                          .stSerial1.stComOut.D[0]  		:= TIIB[PCM A (EP6002-0002)]^COM RxPDO-Map Outputs Channel 1^Data Out 0;
                          .stSerial1.stComOut.D[1]  		:= TIIB[PCM A (EP6002-0002)]^COM RxPDO-Map Outputs Channel 1^Data Out 1;
                          .stSerial1.stComOut.D[2]  		:= TIIB[PCM A (EP6002-0002)]^COM RxPDO-Map Outputs Channel 1^Data Out 2;
                          .stSerial1.stComOut.D[3]  		:= TIIB[PCM A (EP6002-0002)]^COM RxPDO-Map Outputs Channel 1^Data Out 3;
                          .stSerial1.stComOut.D[4]  		:= TIIB[PCM A (EP6002-0002)]^COM RxPDO-Map Outputs Channel 1^Data Out 4;
                          .stSerial1.stComOut.D[5]  		:= TIIB[PCM A (EP6002-0002)]^COM RxPDO-Map Outputs Channel 1^Data Out 5;
                          .stSerial1.stComOut.D[6]  		:= TIIB[PCM A (EP6002-0002)]^COM RxPDO-Map Outputs Channel 1^Data Out 6;
                          .stSerial1.stComOut.D[7]  		:= TIIB[PCM A (EP6002-0002)]^COM RxPDO-Map Outputs Channel 1^Data Out 7;
                          .stSerial1.stComOut.D[8]  		:= TIIB[PCM A (EP6002-0002)]^COM RxPDO-Map Outputs Channel 1^Data Out 8;
                          .stSerial1.stComOut.D[9]  		:= TIIB[PCM A (EP6002-0002)]^COM RxPDO-Map Outputs Channel 1^Data Out 9;
                          .stSerial1.stComOut.D[10]  		:= TIIB[PCM A (EP6002-0002)]^COM RxPDO-Map Outputs Channel 1^Data Out 10;
                          .stSerial1.stComOut.D[11]  		:= TIIB[PCM A (EP6002-0002)]^COM RxPDO-Map Outputs Channel 1^Data Out 11;
                          .stSerial1.stComOut.D[12]  		:= TIIB[PCM A (EP6002-0002)]^COM RxPDO-Map Outputs Channel 1^Data Out 12;
                          .stSerial1.stComOut.D[13]  		:= TIIB[PCM A (EP6002-0002)]^COM RxPDO-Map Outputs Channel 1^Data Out 13;
                          .stSerial1.stComOut.D[14]  		:= TIIB[PCM A (EP6002-0002)]^COM RxPDO-Map Outputs Channel 1^Data Out 14;
                          .stSerial1.stComOut.D[15]  		:= TIIB[PCM A (EP6002-0002)]^COM RxPDO-Map Outputs Channel 1^Data Out 15;
                          .stSerial1.stComOut.D[16]  		:= TIIB[PCM A (EP6002-0002)]^COM RxPDO-Map Outputs Channel 1^Data Out 16;
                          .stSerial1.stComOut.D[17]  		:= TIIB[PCM A (EP6002-0002)]^COM RxPDO-Map Outputs Channel 1^Data Out 17;
                          .stSerial1.stComOut.D[18]  		:= TIIB[PCM A (EP6002-0002)]^COM RxPDO-Map Outputs Channel 1^Data Out 18;
                          .stSerial1.stComOut.D[19]  		:= TIIB[PCM A (EP6002-0002)]^COM RxPDO-Map Outputs Channel 1^Data Out 19;
                          .stSerial1.stComOut.D[20]  		:= TIIB[PCM A (EP6002-0002)]^COM RxPDO-Map Outputs Channel 1^Data Out 20;
                          .stSerial1.stComOut.D[21]  		:= TIIB[PCM A (EP6002-0002)]^COM RxPDO-Map Outputs Channel 1^Data Out 21;

                          .stSerial2.stComOut.D[0]  		:= TIIB[PCM A (EP6002-0002)]^COM RxPDO-Map Outputs Channel 2^Data Out 0;
                          .stSerial2.stComOut.D[1]  		:= TIIB[PCM A (EP6002-0002)]^COM RxPDO-Map Outputs Channel 2^Data Out 1;
                          .stSerial2.stComOut.D[2]  		:= TIIB[PCM A (EP6002-0002)]^COM RxPDO-Map Outputs Channel 2^Data Out 2;
                          .stSerial2.stComOut.D[3]  		:= TIIB[PCM A (EP6002-0002)]^COM RxPDO-Map Outputs Channel 2^Data Out 3;
                          .stSerial2.stComOut.D[4]  		:= TIIB[PCM A (EP6002-0002)]^COM RxPDO-Map Outputs Channel 2^Data Out 4;
                          .stSerial2.stComOut.D[5]  		:= TIIB[PCM A (EP6002-0002)]^COM RxPDO-Map Outputs Channel 2^Data Out 5;
                          .stSerial2.stComOut.D[6]  		:= TIIB[PCM A (EP6002-0002)]^COM RxPDO-Map Outputs Channel 2^Data Out 6;
                          .stSerial2.stComOut.D[7]  		:= TIIB[PCM A (EP6002-0002)]^COM RxPDO-Map Outputs Channel 2^Data Out 7;
                          .stSerial2.stComOut.D[8]  		:= TIIB[PCM A (EP6002-0002)]^COM RxPDO-Map Outputs Channel 2^Data Out 8;
                          .stSerial2.stComOut.D[9]  		:= TIIB[PCM A (EP6002-0002)]^COM RxPDO-Map Outputs Channel 2^Data Out 9;
                          .stSerial2.stComOut.D[10] 	 	:= TIIB[PCM A (EP6002-0002)]^COM RxPDO-Map Outputs Channel 2^Data Out 10;
                          .stSerial2.stComOut.D[11] 	 	:= TIIB[PCM A (EP6002-0002)]^COM RxPDO-Map Outputs Channel 2^Data Out 11;
                          .stSerial2.stComOut.D[12] 	 	:= TIIB[PCM A (EP6002-0002)]^COM RxPDO-Map Outputs Channel 2^Data Out 12;
                          .stSerial2.stComOut.D[13] 	 	:= TIIB[PCM A (EP6002-0002)]^COM RxPDO-Map Outputs Channel 2^Data Out 13;
                          .stSerial2.stComOut.D[14] 	 	:= TIIB[PCM A (EP6002-0002)]^COM RxPDO-Map Outputs Channel 2^Data Out 14;
                          .stSerial2.stComOut.D[15] 	 	:= TIIB[PCM A (EP6002-0002)]^COM RxPDO-Map Outputs Channel 2^Data Out 15;
                          .stSerial2.stComOut.D[16] 	 	:= TIIB[PCM A (EP6002-0002)]^COM RxPDO-Map Outputs Channel 2^Data Out 16;
                          .stSerial2.stComOut.D[17] 	 	:= TIIB[PCM A (EP6002-0002)]^COM RxPDO-Map Outputs Channel 2^Data Out 17;
                          .stSerial2.stComOut.D[18] 	 	:= TIIB[PCM A (EP6002-0002)]^COM RxPDO-Map Outputs Channel 2^Data Out 18;
                          .stSerial2.stComOut.D[19] 	 	:= TIIB[PCM A (EP6002-0002)]^COM RxPDO-Map Outputs Channel 2^Data Out 19;
                          .stSerial2.stComOut.D[20] 	 	:= TIIB[PCM A (EP6002-0002)]^COM RxPDO-Map Outputs Channel 2^Data Out 20;
                          .stSerial2.stComOut.D[21] 	 	:= TIIB[PCM A (EP6002-0002)]^COM RxPDO-Map Outputs Channel 2^Data Out 21;
'}
PCMA : FB_PressureControlModule;

{attribute 'pytmc' := 'pv: XCS:SDS:PCM:B'}
{attribute 'TcLinkTo' := '.stPropAir1.i_iPressRB 	:= TIIB[PCM B (EP4374-0002)]^AI Inputs Channel 1^Value;
                          .stPropAir2.i_iPressRB 	:= TIIB[PCM B (EP4374-0002)]^AI Inputs Channel 2^Value;
                          .stPropAir1.q_iPressCt 	:= TIIB[PCM B (EP4374-0002)]^AO Outputs Channel 3^Analog output;
                          .stPropAir2.q_iPressCt 	:= TIIB[PCM B (EP4374-0002)]^AO Outputs Channel 4^Analog output;
                          .stSerial1.stComIn.Status := TIIB[PCM B (EP6002-0002)]^COM TxPDO-Map Inputs Channel 1^Status;
                          .stSerial2.stComIn.Status := TIIB[PCM B (EP6002-0002)]^COM TxPDO-Map Inputs Channel 2^Status;
                          .stSerial1.stComOut.Ctrl 	:= TIIB[PCM B (EP6002-0002)]^COM RxPDO-Map Outputs Channel 1^Ctrl;
                          .stSerial2.stComOut.Ctrl 	:= TIIB[PCM B (EP6002-0002)]^COM RxPDO-Map Outputs Channel 2^Ctrl;
                          .stBaseIO.i_SyncUnitWC 	:= TIIB[PCM B (EP1111)]^WcState^WcState;
'}
PCMB : FB_PressureControlModule;

{attribute 'pytmc' := 'pv: XCS:SDS:PCM:C'}
{attribute 'TcLinkTo' := '.stPropAir1.i_iPressRB 	:= TIIB[PCM C (EP4374-0002)]^AI Inputs Channel 1^Value;
                          .stPropAir2.i_iPressRB 	:= TIIB[PCM C (EP4374-0002)]^AI Inputs Channel 2^Value;
                          .stPropAir1.q_iPressCt 	:= TIIB[PCM C (EP4374-0002)]^AO Outputs Channel 3^Analog output;
                          .stPropAir2.q_iPressCt 	:= TIIB[PCM C (EP4374-0002)]^AO Outputs Channel 4^Analog output;
                          .stSerial1.stComIn.Status := TIIB[PCM C (EP6002-0002)]^COM TxPDO-Map Inputs Channel 1^Status;
                          .stSerial2.stComIn.Status := TIIB[PCM C (EP6002-0002)]^COM TxPDO-Map Inputs Channel 2^Status;
                          .stSerial1.stComOut.Ctrl 	:= TIIB[PCM C (EP6002-0002)]^COM RxPDO-Map Outputs Channel 1^Ctrl;
                          .stSerial2.stComOut.Ctrl 	:= TIIB[PCM C (EP6002-0002)]^COM RxPDO-Map Outputs Channel 2^Ctrl;
                          .stBaseIO.i_SyncUnitWC 	:= TIIB[PCM C (EP1111)]^WcState^WcState;
                          '}
PCMC : FB_PressureControlModule;

//Pumpless recirc
{attribute 'pytmc' := 'pv: XCS:SDS:PCM:D'}
{attribute 'TcLinkTo' := '.stPropAir1.i_iPressRB 	:= TIIB[PCM D (EP4374-0002)]^AI Inputs Channel 1^Value;
                          .stPropAir2.i_iPressRB 	:= TIIB[PCM D (EP4374-0002)]^AI Inputs Channel 2^Value;
                          .stPropAir1.q_iPressCt 	:= TIIB[PCM D (EP4374-0002)]^AO Outputs Channel 3^Analog output;
                          .stPropAir2.q_iPressCt 	:= TIIB[PCM D (EP4374-0002)]^AO Outputs Channel 4^Analog output;
                          .stSerial1.stComIn.Status := TIIB[PCM D (EP6002-0002)]^COM TxPDO-Map Inputs Channel 1^Status;
                          .stSerial2.stComIn.Status := TIIB[PCM D (EP6002-0002)]^COM TxPDO-Map Inputs Channel 2^Status;
                          .stSerial1.stComOut.Ctrl 	:= TIIB[PCM D (EP6002-0002)]^COM RxPDO-Map Outputs Channel 1^Ctrl;
                          .stSerial2.stComOut.Ctrl 	:= TIIB[PCM D (EP6002-0002)]^COM RxPDO-Map Outputs Channel 2^Ctrl;
                          .stBaseIO.i_SyncUnitWC 	:= TIIB[PCM D (EP1111)]^WcState^WcState;
                          '}
PCMD : FB_PressureControlModule;

{attribute 'pytmc' := 'pv: XCS:SDS:PCM:E'}
{attribute 'TcLinkTo' := '.stPropAir1.i_iPressRB 	:= TIIB[Box 63 (EP4374-0002)]^AI Inputs Channel 1^Value;
                          .stPropAir2.i_iPressRB 	:= TIIB[Box 63 (EP4374-0002)]^AI Inputs Channel 2^Value;
                          .stPropAir1.q_iPressCt 	:= TIIB[Box 63 (EP4374-0002)]^AO Outputs Channel 3^Analog output;
                          .stPropAir2.q_iPressCt 	:= TIIB[Box 63 (EP4374-0002)]^AO Outputs Channel 4^Analog output;
                          .stBaseIO.i_SyncUnitWC 	:= TIIB[Box 28 (EP1111)]^WcState^WcState;
                          '}
PCME : FB_PressureControlModule;

{attribute 'pytmc' := 'pv: XCS:SDS:MAN'}
{attribute 'TcLinkTo' := '.stValve[1].qxDO := TIIB[Gas_Mani_ValveCtrl (EP2338-0001)]^Channel 9^Output;
                          .stValve[1].ixOPN := TIIB[Gas_Mani_ValveRbk (EP2338-0001)]^Channel 1^Input;
                          .stValve[2].qxDO := TIIB[Gas_Mani_ValveCtrl (EP2338-0001)]^Channel 10^Output;
                          .stValve[2].ixOPN := TIIB[Gas_Mani_ValveRbk (EP2338-0001)]^Channel 2^Input;
                          .stValve[3].qxDO := TIIB[Gas_Mani_ValveCtrl (EP2338-0001)]^Channel 11^Output;
                          .stValve[3].ixOPN := TIIB[Gas_Mani_ValveRbk (EP2338-0001)]^Channel 3^Input;
                          .stValve[4].qxDO := TIIB[Gas_Mani_ValveCtrl (EP2338-0001)]^Channel 12^Output;
                          .stValve[4].ixOPN := TIIB[Gas_Mani_ValveRbk (EP2338-0001)]^Channel 4^Input;
                          .stValve[5].qxDO := TIIB[Gas_Mani_ValveCtrl (EP2338-0001)]^Channel 13^Output;
                          .stValve[5].ixOPN := TIIB[Gas_Mani_ValveRbk (EP2338-0001)]^Channel 5^Input;
                          .stValve[6].qxDO := TIIB[Gas_Mani_ValveCtrl (EP2338-0001)]^Channel 14^Output;
                          .stValve[6].ixOPN := TIIB[Gas_Mani_ValveRbk (EP2338-0001)]^Channel 6^Input;
                          .stValve[7].qxDO := TIIB[Gas_Mani_ValveCtrl (EP2338-0001)]^Channel 15^Output;
                          .stValve[7].ixOPN := TIIB[Gas_Mani_ValveRbk (EP2338-0001)]^Channel 7^Input;
                          .stBaseIO.i_SyncUnitWC :=	TIID^MAIN (EtherCAT)^Gas_Mani (EP1111)^WcState^WcState;
'}
GasMan : FB_GasManifold;

{attribute 'pytmc' := 'pv: XCS:SDS:MFM:A'}
{attribute 'TcLinkTo' := '.stMFM.i_rFlow := TIID^MAIN (EtherCAT)^Bronkhorst MFM A^TxPDO Map^fMeasure;
                          .stMFM.q_rSetpoint := TIID^MAIN (EtherCAT)^Bronkhorst MFM A^RxPDO Map^fSetpoint;
'}
BronkhorstA : FB_BronkhorstMFM;

{attribute 'pytmc' := 'pv: XCS:SDS:MFM:B'}
{attribute 'TcLinkTo' := '.stMFM.i_rFlow 		:= TIIB[Bronkhorst MFM B]^TxPDO Map^fMeasure;
                          .stMFM.q_rSetpoint 	:=  TIIB[Bronkhorst MFM B]^RxPDO Map^fSetpoint;
'}
BronkhorstB : FB_BronkhorstMFM;

{attribute 'pytmc' := 'pv: XCS:SDS:MFM:C'}
{attribute 'TcLinkTo' := '.stMFM.i_rFlow := TIID^MAIN (EtherCAT)^Bronkhorst MFM C^TxPDO Map^fMeasure;
                          .stMFM.q_rSetpoint := TIID^MAIN (EtherCAT)^Bronkhorst MFM C^RxPDO Map^fSetpoint;
'}
BronkhorstC : FB_BronkhorstMFM;

{attribute 'pytmc' := 'pv: XCS:SDS:MFM:D'}
{attribute 'TcLinkTo' := '.stMFM.i_rFlow := TIID^MAIN (EtherCAT)^Bronkhorst MFM D^TxPDO Map^fMeasure;
                          .stMFM.q_rSetpoint := TIID^MAIN (EtherCAT)^Bronkhorst MFM D^RxPDO Map^fSetpoint;
'}
BronkhorstD : FB_BronkhorstMFM;

{attribute 'pytmc' := 'pv: XCS:SDS:SPR:A'}
{attribute 'TcLinkTo' := '.q_xDO1 := TIIB[Solenoid Pair A Digital IO (EP2338-0001)]^Channel 9^Output;
                          .q_xDO2 := TIIB[Solenoid Pair A Digital IO (EP2338-0001)]^Channel 10^Output;
'}
SolenoidPairA : FB_SolenoidPair;


END_VAR

// ---- POUs/MAIN.TcPOU
PROGRAM MAIN
VAR

END_VAR

M3SelectorA();
M3SelectorB();
M3SelectorC();
M3SelectorD();
PCMA();
PCMB();
PCMC();
PCMD();
GasMan();
BronkhorstA();
BronkhorstB();
BronkhorstC();
BronkhorstD();
SolenoidPairA();

PRG_RCC();

(* Following execution of all the programs, set the first pass false *)
g_xFirstPass := FALSE;

END_PROGRAM

// ---- POUs/PRG_RCC.TcPOU
PROGRAM PRG_RCC
VAR

    {attribute 'pytmc' :=' pv: XCS:RCC:01'}
    stRCC_CTL_SIM : ST_RCC;
    fbRCC_SIM 	  : FB_RCC;

    {attribute 'pytmc' :=' pv: XCS:RCC:02'}
    stRCC_CTL_HPLC : ST_RCC;
    fbRCC_HPLC 	  : FB_RCC;

    RCC_GCP_01_dummy : ST_VG;
    xSystemOverrideMode_RCC : BOOL := FALSE;
END_VAR

// dummy gauge is used to allow for RCC withough gauge interlock
RCC_GCP_01_dummy.xPRESS_OK := TRUE;
stRCC_CTL_HPLC.RCC_VRC_03_OPEN_OK := TRUE;

fbRCC_SIM( stRCC_VRC_01:= RCC_VRC_01.iq_stValve,
    stRCC_VRC_02 := RCC_VRC_02.iq_stValve,
    stRCC_VRC_03 := RCC_VRC_03.iq_stValve,
    stRCC_VRC_04 := RCC_VRC_04.iq_stValve,
    stRCC_GCP_01 := RCC_GCP_01_dummy,
    stRCC_CTL := stRCC_CTL_SIM
);


fbRCC_HPLC( stRCC_VRC_01:= RCC_VRC_05.iq_stValve,
    stRCC_VRC_02 := RCC_VRC_06.iq_stValve,
    stRCC_VRC_03 := RCC_VRC_07.iq_stValve,
    stRCC_VRC_04 := RCC_VRC_08.iq_stValve,
    stRCC_GCP_01 := RCC_GCP_01_dummy,
    stRCC_CTL := stRCC_CTL_HPLC
);

RCC_VRC_01(i_xExtILK_OK := stRCC_CTL_SIM.RCC_VRC_01_OPEN_OK,
                i_xOverrideMode := xSystemOverrideMode_RCC,
                 iq_stValve=> );

RCC_VRC_02(i_xExtILK_OK := stRCC_CTL_SIM.RCC_VRC_02_OPEN_OK,
                i_xOverrideMode := xSystemOverrideMode_RCC,
                 iq_stValve=> );
RCC_VRC_03(i_xExtILK_OK := stRCC_CTL_SIM.RCC_VRC_03_OPEN_OK,
                i_xOverrideMode := xSystemOverrideMode_RCC,
                 iq_stValve=> );

RCC_VRC_04(i_xExtILK_OK := stRCC_CTL_SIM.RCC_VRC_04_OPEN_OK,
                i_xOverrideMode := xSystemOverrideMode_RCC,
                 iq_stValve=> );
RCC_VRC_05(i_xExtILK_OK := stRCC_CTL_HPLC.RCC_VRC_01_OPEN_OK,
                i_xOverrideMode := xSystemOverrideMode_RCC,
                 iq_stValve=> );

RCC_VRC_06(i_xExtILK_OK := stRCC_CTL_HPLC.RCC_VRC_02_OPEN_OK,
                i_xOverrideMode := xSystemOverrideMode_RCC,
                 iq_stValve=> );
RCC_VRC_07(i_xExtILK_OK := stRCC_CTL_HPLC.RCC_VRC_03_OPEN_OK,
                i_xOverrideMode := xSystemOverrideMode_RCC,
                 iq_stValve=> );

RCC_VRC_08(i_xExtILK_OK := stRCC_CTL_HPLC.RCC_VRC_04_OPEN_OK,
                i_xOverrideMode := xSystemOverrideMode_RCC,
                 iq_stValve=> );

END_PROGRAM
